% RSLogix 500 project Pump Protection.RSS, saved by version 8.30.00.16 %
PROJECT "UNTITLED"    % processor: Bul.1763 MicroLogix 1100 Series B %

PROGRAM FILES
  LAD 2 "MAIN"  4 rungs
  LAD 3 "DIGITAL IO"  10 rungs
  LAD 4 "ALARMS"  11 rungs
  LAD 5 "CONTROLS"  10 rungs

DATA FILES
  O0 OUTPUT  5 elements
  I1 INPUT  7 elements
  S2 STATUS  66 elements
  B3 BINARY  2 elements
  T4 TIMER  4 elements
  C5 COUNTER  1 elements
  R6 CONTROL  1 elements
  N7 INTEGER  3 elements
  F8 FLOAT  1 elements

LADDER 2 "MAIN"
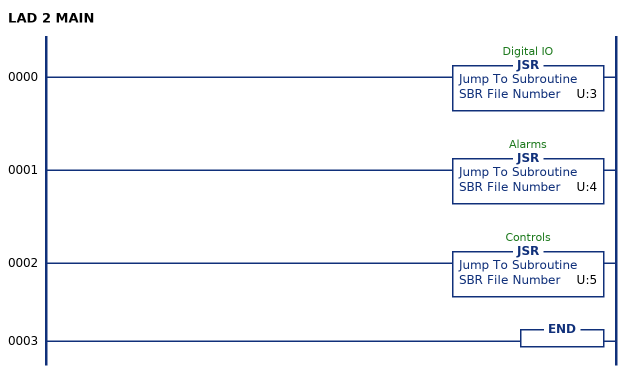
% Rung: 0 %
SOR JSR U:3 EOR
%   U:3  "Digital IO" %
% Rung: 1 %
SOR JSR U:4 EOR
%   U:4  "Alarms" %
% Rung: 2 %
SOR JSR U:5 EOR
%   U:5  "Controls" %
% Rung: 3 %
SOR END EOR

LADDER 3 "DIGITAL IO"
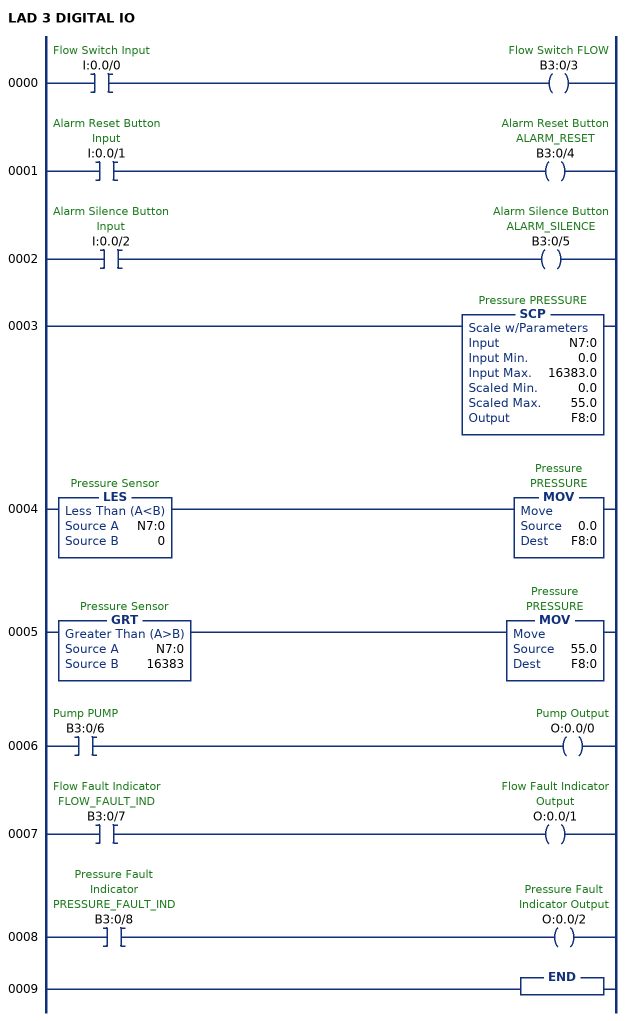
% Rung: 0 %
SOR XIC I:0.0/0 OTE B3:0/3 EOR
%   I:0.0/0  "Flow Switch Input" %
%   B3:0/3  FLOW  "Flow Switch" %
% Rung: 1 %
SOR XIC I:0.0/1 OTE B3:0/4 EOR
%   I:0.0/1  "Alarm Reset Button Input" %
%   B3:0/4  ALARM_RESET  "Alarm Reset Button" %
% Rung: 2 %
SOR XIC I:0.0/2 OTE B3:0/5 EOR
%   I:0.0/2  "Alarm Silence Button Input" %
%   B3:0/5  ALARM_SILENCE  "Alarm Silence Button" %
% Rung: 3 %
SOR SCP N7:0 0.0 16383.0 0.0 55.0 F8:0 EOR
%   N7:0  "Pressure Sensor" %
%   F8:0  PRESSURE  "Pressure" %
% Rung: 4 %
SOR LES N7:0 0 MOV 0.0 F8:0 EOR
%   N7:0  "Pressure Sensor" %
%   F8:0  PRESSURE  "Pressure" %
% Rung: 5 %
SOR GRT N7:0 16383 MOV 55.0 F8:0 EOR
%   N7:0  "Pressure Sensor" %
%   F8:0  PRESSURE  "Pressure" %
% Rung: 6 %
SOR XIC B3:0/6 OTE O:0.0/0 EOR
%   B3:0/6  PUMP  "Pump" %
%   O:0.0/0  "Pump Output" %
% Rung: 7 %
SOR XIC B3:0/7 OTE O:0.0/1 EOR
%   B3:0/7  FLOW_FAULT_IND  "Flow Fault Indicator" %
%   O:0.0/1  "Flow Fault Indicator Output" %
% Rung: 8 %
SOR XIC B3:0/8 OTE O:0.0/2 EOR
%   B3:0/8  PRESSURE_FAULT_IND  "Pressure Fault Indicator" %
%   O:0.0/2  "Pressure Fault Indicator Output" %
% Rung: 9 %
SOR END EOR

LADDER 4 "ALARMS"
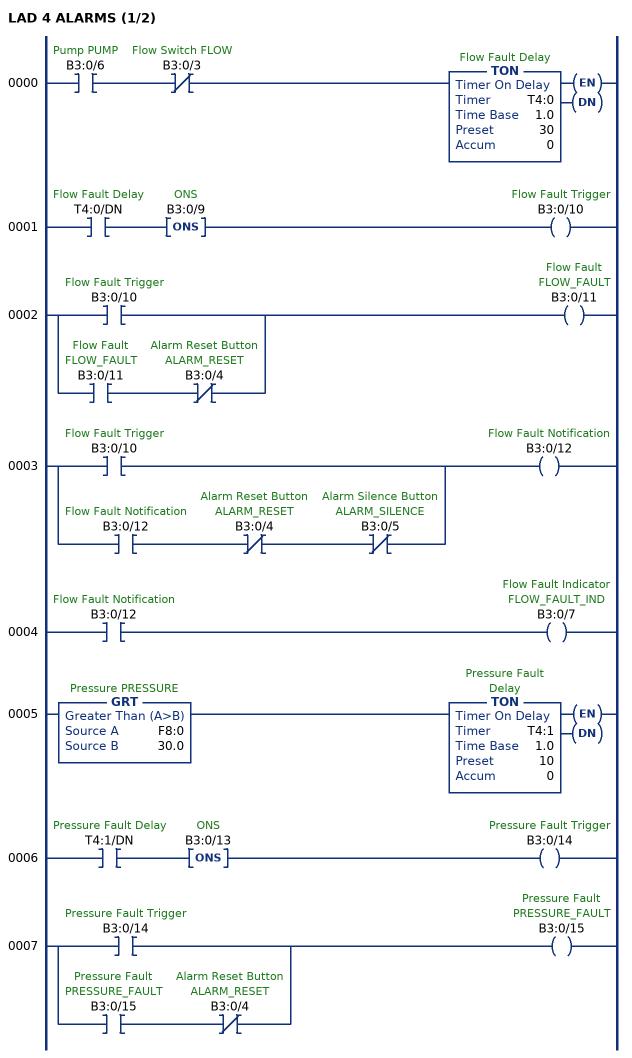
% Rung: 0 %
SOR XIC B3:0/6 XIO B3:0/3 TON T4:0 1.0 30 0 EOR
%   B3:0/6  PUMP  "Pump" %
%   B3:0/3  FLOW  "Flow Switch" %
%   T4:0  "Flow Fault Delay" %
% Rung: 1 %
SOR XIC T4:0/DN ONS B3:0/9 OTE B3:0/10 EOR
%   T4:0  "Flow Fault Delay" %
%   B3:0/9  "ONS" %
%   B3:0/10  "Flow Fault Trigger" %
% Rung: 2 %
SOR BST XIC B3:0/10 NXB XIC B3:0/11 XIO B3:0/4 BND OTE B3:0/11 EOR
%   B3:0/10  "Flow Fault Trigger" %
%   B3:0/11  FLOW_FAULT  "Flow Fault" %
%   B3:0/4  ALARM_RESET  "Alarm Reset Button" %
% Rung: 3 %
SOR BST XIC B3:0/10 NXB XIC B3:0/12 XIO B3:0/4 XIO B3:0/5 BND OTE B3:0/12 EOR
%   B3:0/10  "Flow Fault Trigger" %
%   B3:0/12  "Flow Fault Notification" %
%   B3:0/4  ALARM_RESET  "Alarm Reset Button" %
%   B3:0/5  ALARM_SILENCE  "Alarm Silence Button" %
% Rung: 4 %
SOR XIC B3:0/12 OTE B3:0/7 EOR
%   B3:0/12  "Flow Fault Notification" %
%   B3:0/7  FLOW_FAULT_IND  "Flow Fault Indicator" %
% Rung: 5 %
SOR GRT F8:0 30.0 TON T4:1 1.0 10 0 EOR
%   F8:0  PRESSURE  "Pressure" %
%   T4:1  "Pressure Fault Delay" %
% Rung: 6 %
SOR XIC T4:1/DN ONS B3:0/13 OTE B3:0/14 EOR
%   T4:1  "Pressure Fault Delay" %
%   B3:0/13  "ONS" %
%   B3:0/14  "Pressure Fault Trigger" %
% Rung: 7 %
SOR BST XIC B3:0/14 NXB XIC B3:0/15 XIO B3:0/4 BND OTE B3:0/15 EOR
%   B3:0/14  "Pressure Fault Trigger" %
%   B3:0/15  PRESSURE_FAULT  "Pressure Fault" %
%   B3:0/4  ALARM_RESET  "Alarm Reset Button" %

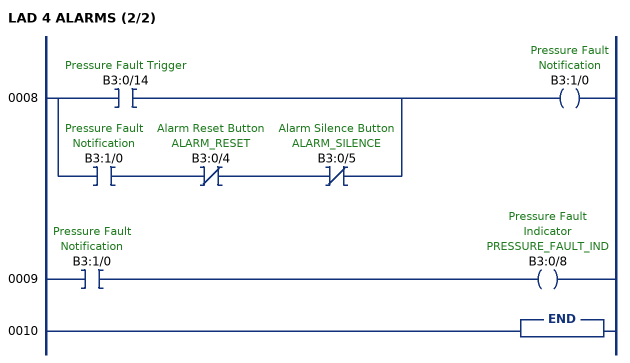
% Rung: 8 %
SOR BST XIC B3:0/14 NXB XIC B3:1/0 XIO B3:0/4 XIO B3:0/5 BND OTE B3:1/0 EOR
%   B3:0/14  "Pressure Fault Trigger" %
%   B3:1/0  "Pressure Fault Notification" %
%   B3:0/4  ALARM_RESET  "Alarm Reset Button" %
%   B3:0/5  ALARM_SILENCE  "Alarm Silence Button" %
% Rung: 9 %
SOR XIC B3:1/0 OTE B3:0/8 EOR
%   B3:1/0  "Pressure Fault Notification" %
%   B3:0/8  PRESSURE_FAULT_IND  "Pressure Fault Indicator" %
% Rung: 10 %
SOR END EOR

LADDER 5 "CONTROLS"
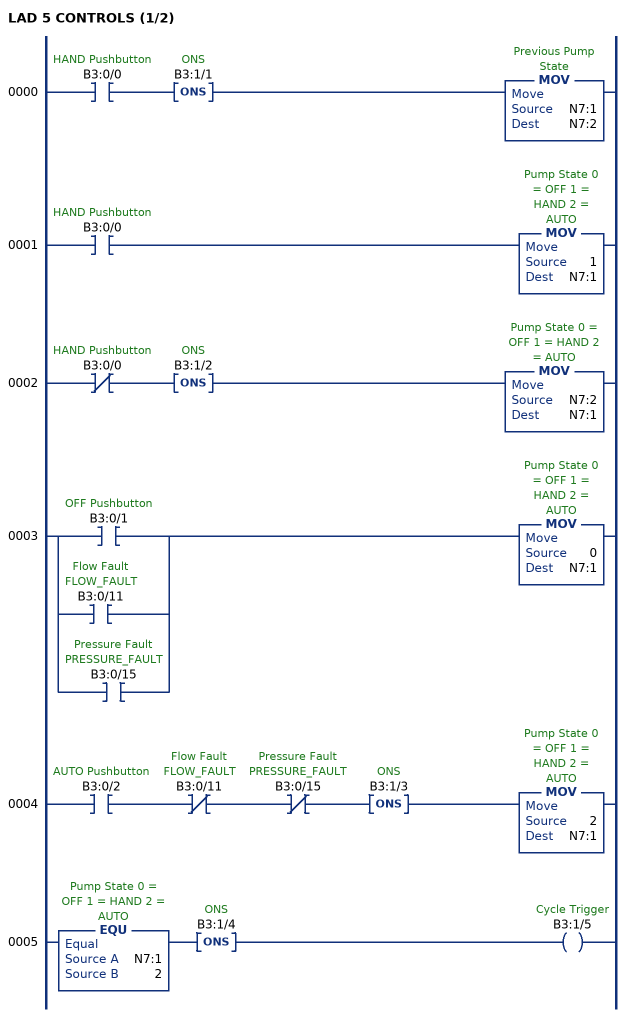
% Rung: 0 %
SOR XIC B3:0/0 ONS B3:1/1 MOV N7:1 N7:2 EOR
%   B3:0/0  "HAND Pushbutton" %
%   B3:1/1  "ONS" %
%   N7:1  "Pump State 0 = OFF 1 = HAND 2 = AUTO" %
%   N7:2  "Previous Pump State" %
% Rung: 1 %
SOR XIC B3:0/0 MOV 1 N7:1 EOR
%   B3:0/0  "HAND Pushbutton" %
%   N7:1  "Pump State 0 = OFF 1 = HAND 2 = AUTO" %
% Rung: 2 %
SOR XIO B3:0/0 ONS B3:1/2 MOV N7:2 N7:1 EOR
%   B3:0/0  "HAND Pushbutton" %
%   B3:1/2  "ONS" %
%   N7:2  "Previous Pump State" %
%   N7:1  "Pump State 0 = OFF 1 = HAND 2 = AUTO" %
% Rung: 3 %
SOR BST XIC B3:0/1 NXB XIC B3:0/11 NXB XIC B3:0/15 BND MOV 0 N7:1 EOR
%   B3:0/1  "OFF Pushbutton" %
%   B3:0/11  FLOW_FAULT  "Flow Fault" %
%   B3:0/15  PRESSURE_FAULT  "Pressure Fault" %
%   N7:1  "Pump State 0 = OFF 1 = HAND 2 = AUTO" %
% Rung: 4 %
SOR XIC B3:0/2 XIO B3:0/11 XIO B3:0/15 ONS B3:1/3 MOV 2 N7:1 EOR
%   B3:0/2  "AUTO Pushbutton" %
%   B3:0/11  FLOW_FAULT  "Flow Fault" %
%   B3:0/15  PRESSURE_FAULT  "Pressure Fault" %
%   B3:1/3  "ONS" %
%   N7:1  "Pump State 0 = OFF 1 = HAND 2 = AUTO" %
% Rung: 5 %
SOR EQU N7:1 2 ONS B3:1/4 OTE B3:1/5 EOR
%   N7:1  "Pump State 0 = OFF 1 = HAND 2 = AUTO" %
%   B3:1/4  "ONS" %
%   B3:1/5  "Cycle Trigger" %

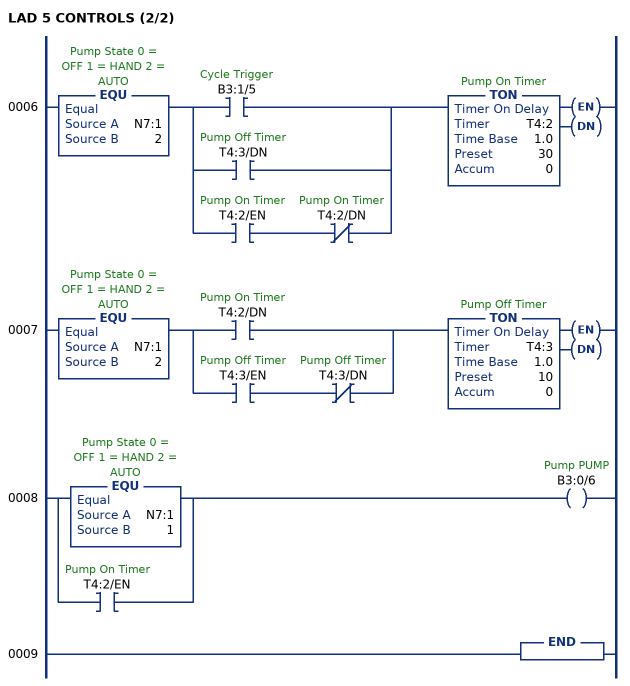
% Rung: 6 %
SOR EQU N7:1 2 BST XIC B3:1/5 NXB XIC T4:3/DN NXB XIC T4:2/EN XIO T4:2/DN BND TON T4:2 1.0 30 0 EOR
%   N7:1  "Pump State 0 = OFF 1 = HAND 2 = AUTO" %
%   B3:1/5  "Cycle Trigger" %
%   T4:3  "Pump Off Timer" %
%   T4:2  "Pump On Timer" %
% Rung: 7 %
SOR EQU N7:1 2 BST XIC T4:2/DN NXB XIC T4:3/EN XIO T4:3/DN BND TON T4:3 1.0 10 0 EOR
%   N7:1  "Pump State 0 = OFF 1 = HAND 2 = AUTO" %
%   T4:2  "Pump On Timer" %
%   T4:3  "Pump Off Timer" %
% Rung: 8 %
SOR BST EQU N7:1 1 NXB XIC T4:2/EN BND OTE B3:0/6 EOR
%   N7:1  "Pump State 0 = OFF 1 = HAND 2 = AUTO" %
%   T4:2  "Pump On Timer" %
%   B3:0/6  PUMP  "Pump" %
% Rung: 9 %
SOR END EOR

DATA TABLE (non-zero values as saved)
DATA T4
% .PRE .ACC %
% T4:0 % 30 0
% T4:1 % 10 0
% T4:2 % 30 0
% T4:3 % 10 0
